# EPICS substitutions: viocs/si_ps/si_psApp/Db/sdp0.substitutions
file "db/individual.db" {
    pattern { family, pos, num }
        { "SDP0", "03M1", "" }
        { "SDP0", "03M2", "" }
        { "SDP0", "07M1", "" }
        { "SDP0", "07M2", "" }
        { "SDP0", "11M1", "" }
        { "SDP0", "11M2", "" }
        { "SDP0", "15M1", "" }
        { "SDP0", "15M2", "" }
        { "SDP0", "19M1", "" }
        { "SDP0", "19M2", "" }
}
